{attribute 'linkalways'} 
{attribute 'no_explicit_call' := 'This FB is a CLASS and must be accessed using methods or properties'}
{attribute 'enable_dynamic_creation'}
FUNCTION_BLOCK FINAL MUL_UDINT EXTENDS Node
VAR
	in1 : _UDINT(0);
	in2 : _UDINT(0);
	out : _UDINT(0);
END_VAR

METHOD PUBLIC Clone : I_Node
VAR
	pNode : POINTER TO MUL_UDINT;
END_VAR
pNode := __NEW(MUL_UDINT);
Clone := pNode^;
END_METHOD

METHOD FB_init : BOOL
VAR_INPUT
	bInitRetains : BOOL; // if TRUE, the retain variables are initialized (warm start / cold start)
	bInCopyCode : BOOL;  // if TRUE, the instance afterwards gets moved into the copy code (online change)
END_VAR
AddInput('in1',THIS^.in1);
AddInput('in2',THIS^.in2);
AddOutput('out', THIS^.out);
END_METHOD

METHOD PROTECTED OnExecute
VAR
END_VAR
out.Value := in1.Value * in2.Value;
END_METHOD

END_FUNCTION_BLOCK

(* stored: Version 1.1.0.1, ProductVersion 3.1.4024.15
   POU MUL_UDINT: Id {6b2b8ddb-4725-421f-b44f-02435ab860ee}, SpecialFunc None
   Folder Constructor: Id {002af86d-616f-4560-b996-2723545c808a}
   Method Clone: Id {31cb1e14-1e83-41e6-a7e9-7310ebdc1400}
   Method FB_init: Id {426ebde2-e925-4eb0-ab8e-577fd2379b66}
   Method OnExecute: Id {455c2f5b-3de6-4426-8b84-1393cae7974d} *)
